// TIA Portal V19 export
DATA_BLOCK "A0302_Rulliera_PERS"   // DB119
// stored: MemoryReserve 100
   VAR RETAIN
      Par : Struct
         Ax { S7_SetPoint := 'True'} : "SpeedMachine_Par";
         Ax_Aut { S7_SetPoint := 'True'} : "A0301_Mach_Speed_Par";
      END_STRUCT;
      IEC_SP : Struct
         FTC_CodaRall : Struct
            TON_PT : Time := T#300MS;
            TOF_PT : Time := T#300MS;
         END_STRUCT;
         FTC_CodaProxIng : Struct
            TON_PT : Time := T#300MS;
            TOF_PT : Time := T#300MS;
         END_STRUCT;
         FTC_Centro : Struct
            TON_PT : Time := T#300MS;
            TOF_PT : Time := T#300MS;
         END_STRUCT;
      END_STRUCT;
   END_VAR
BEGIN
   Par.Ax.Man.VelBwd := 2000.0;
   Par.Ax.Man.VelFwdHigh := 50000.0;
   Par.Ax.Man.VelFwdLow := 20000.0;
   Par.Ax.Man.Acc := 2000.0;
   Par.Ax.Man.Dec := 2000.0;
   Par.Ax.Man.DelayChangeVel := T#200MS;
   Par.Ax_Aut.SemiAut_Vel := 35000.0;
   Par.Ax_Aut.Aut_Vel := 30000.0;
   Par.Ax_Aut.Aut_Acc := 1100.0;
   Par.Ax_Aut.Aut_Dec := 1100.0;
END_DATA_BLOCK
